FUNCTION_BLOCK FlushStartSp (* Basic Function Block Type *)
  (* Standard: 61499-2 *)
  (* Version 0.0, 6/20/2026, Schneider Electric, Template *)
  PACKAGE SE.Nereda;
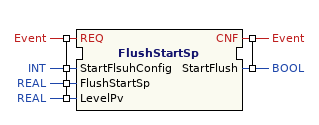
  EVENT_INPUT
    REQ WITH StartFlsuhConfig, FlushStartSp, LevelPv; (* Normal Execution Request *)
  END_EVENT
  EVENT_OUTPUT
    CNF WITH StartFlush; (* Execution Confirmation *)
  END_EVENT
  VAR_INPUT
    StartFlsuhConfig : INT; (* Input event qualifier *)
    FlushStartSp : REAL;
    LevelPv : REAL;
  END_VAR
  VAR_OUTPUT
    StartFlush : BOOL; (* Output event qualifier *)
  END_VAR
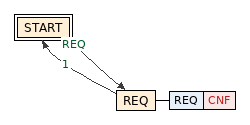
  EC_STATES
    START; (* Initial State *)
    REQ : REQ -> CNF;
  END_STATES
  EC_TRANSITIONS
    START TO REQ := REQ;
    REQ TO START := 1;
  END_TRANSITIONS
  ALGORITHM REQ IN ST: (* Normally executed algorithm *)
;
IF StartFlsuhConfig = 1 THEN
	IF FlushStartSp <= LevelPv THEN
		StartFlush := TRUE;
	ELSE
		StartFlush := FALSE;
	END_IF;
ELSIF StartFlsuhConfig = 2 THEN
	IF FlushStartSp >= LevelPv THEN
		StartFlush := TRUE;
	ELSE
		StartFlush := FALSE;
	END_IF;
END_IF;
  END_ALGORITHM
END_FUNCTION_BLOCK
